Fanuc KAREL source: IO0221.KL

PROGRAM IO0221
%NOLOCKGROUP
ROUTINE RTEST
VAR
L1 : ARRAY[3] OF INTEGER;L2 : XYZWPR
L3 : JOINTPOS9
L4 : POSITION
S1:INTEGER
S2:INTEGER
S3:INTEGER
A:BOOLEAN
B:REAL
BEGIN
--
S1=1
L1[1]=2
A=TRUE
B=1.0
GET_VAR(S3,'*SYSTEM*','$MNUFRAMENUM[1]',S1,S2)
END RTEST
BEGIN
RTEST
END IO0221
